{attribute 'qualified_only'}
{attribute 'strict'}
{attribute 'to_string'}
TYPE E_LogLevel :
(
    Verbose 	:= 1,
    Info  		:= 2,
    Warning  	:= 3,
    Error 		:= 4,
    Critical 	:= 5
);
END_TYPE

(* stored: Version 1.1.0.1
   DUT E_LogLevel: Id {e9ef3f0e-04e3-403f-951a-2d9811693c12} *)
